Staubli VAL3: FC_chrdeal.pgx

program FC_chrdeal(string& x_str[] (dimensions=1))
begin
  //delete all the space " "
  while left(x_str,1)==" "
    x_str=mid(x_str,len(x_str)-1,1)
  endWhile
end
